FUNCTION_BLOCK FB_SimulatedAnaIn_AFO IMPLEMENTS ITF_Schuif_AnaIn_AFO

VAR
	internalState : sint;
END_VAR

{warning 'Add method implementation '}
METHOD get : SINT
get := internalState;
END_METHOD

END_FUNCTION_BLOCK

(* stored: Version 1.1.0.1, ProductVersion 3.1.4026.8
   POU FB_SimulatedAnaIn_AFO: Id {66b4703f-d915-4b8e-9b88-0961f5bebfdd}, SpecialFunc None
   Method get: Id {4a3c7f0e-0e25-4947-87b3-c04699a27469} *)
